// TIA Portal V17 export
// export: Created 2025-06-25T13:13:25.7107653Z, ExportSetting WithDefaults, DisplayName Totally Integrated Automation Portal, DisplayVersion V17 Update 8, DisplayName TIA Portal Openness, DisplayVersion V17 Update 8, DisplayName TIA Portal Version Control Interface, DisplayVersion V17, DisplayName STEP 7 Professional, DisplayVersion V17 Update 8, DisplayName STEP 7 Safety, DisplayVersion V17 Update 6, DisplayName WinCC Advanced, DisplayVersion V17 Update 8
DATA_BLOCK "DB_Application"   // DB9
{ S7_Optimized_Access := 'FALSE' }
VERSION : 0.1
// stored: AutoNumber true, DBAccessibleFromOPCUA true, DBAccessibleFromWebserver true, IsOnlyStoredInLoadMemory false, IsWriteProtectedInAS false
   VAR
      ToHB : Struct
         StartRequest : Bool;
         StopRequest : Bool;
         AlarmAcknowledge : Bool;
         EmergencyStopResetRequest : Bool;
         FastStopRequest : Bool;
         HydrolockProtection : Bool;
         SpareCommand6 : Bool;
         SpareCommand7 : Bool;
         SuperheatManualMode : Bool;
         HeatSinkOutManualMode : Bool;
         PerformanceControlManualMode : Bool;
         OilHeatingRegulatorManualMode : Bool;
         ExpansionValveRegulatorManualMode : Bool;
         PinchRegulatorManualMode : Bool;
         SpareManualMode6 : Bool;
         SpareManualMode7 : Bool;
         PumaCommOk : Bool;   // 1 = communication OK, 0 = communication dead
         HeatSourceOk : Bool;   // 1 = Source ready, 0 = source not ready
         HeatSinkOk : Bool;   // 1 = Sink ready, 0 = sink not ready
         SpareGroup2Command3 : Bool;
         SpareGroup2Command4 : Bool;
         SpareGroup2Command5 : Bool;
         SpareGroup2Command6 : Bool;
         SpareGroup2Command7 : Bool;
         SpareGroup3Command0 : Bool;
         SpareGroup3Command1 : Bool;
         SpareGroup3Command2 : Bool;
         SpareGroup3Command3 : Bool;
         SpareGroup3Command4 : Bool;
         SpareGroup3Command5 : Bool;
         SpareGroup3Command6 : Bool;
         SpareGroup3Command7 : Bool;
         SuperheatManualValue : Real;
         HeatSinkOutManualValue : Real;
         PerformanceControlManualValue : Real;
         OilHeatingManualValue : Real;
         ExpansionValveManualValue : Real;
         PinchManualValue : Real;
         HeatboosterSetpoint : Real;
         RegulationTarget : Int;
         LivenessCounter : UInt;
         HBL_HCV_514_A1 : Real;   // If externally controlled
         HBL_HCV_548_A1 : Real;   // If externally controlled
         HBL_TT_546 : Real;   // If externally controlled
         HBL_PT_547 : Real;   // If externally controlled
         HBL_HCV_515_A1 : Real;   // If externally controlled
         HBL_TT_901 : Real;   // If externally controlled
         HBL_PT_902 : Real;   // If externally controlled
         HBL_TT_512 : Real;   // If externally controlled
         HBL_PT_511 : Real;   // If externally controlled
         HBL_PT_519 : Real;   // If externally controlled
         HBL_TT_518 : Real;   // If externally controlled
      END_STRUCT;
      FromHB : Struct
         EmergencyStop : Bool;
         OilHeatersGroup1 : Bool;
         OilHeatersGroup2 : Bool;
         HBL_SC_01_Ready : Bool;
         HBL_SC_01_Run : Bool;
         HBL_SC_01_Tripped : Bool;
         HBL_SC_02_Ready : Bool;
         HBL_SC_02_Run : Bool;
         HBL_SC_02_Tripped : Bool;
         HBL_SC_10_Ready : Bool;
         HBL_SC_10_Run : Bool;
         HBL_SC_10_Tripped : Bool;
         HBL_HV_630 : Bool;
         HBL_HV_631 : Bool;
         HBL_HV_860 : Bool;
         HBL_HV_861 : Bool;
         HBL_HV_114 : Bool;
         HBL_HV_115 : Bool;
         CPC_P_01 : Bool;
         SSC_P_01 : Bool;
         SSC_F_01 : Bool;
         SSC_P_02 : Bool;
         HBL_LS_01 : Bool;
         HBL_LS_02 : Bool;
         HBL_HV_112 : Bool;
         HBL_HV_113 : Bool;
         HBL_LSH_62 : Bool;
         HBL_LSL_63 : Bool;
         HBL_LSH_64 : Bool;
         HBL_LSL_864 : Bool;
         HBL_LS_632 : Bool;
         HBL_LS_633 : Bool;
         HBL_SC_03_Ready : Bool;
         HBL_SC_03_Run : Bool;
         HBL_SC_03_Tripped : Bool;
         HBL_HCV_514_Force : Bool;
         HBL_HCV_548_Force : Bool;
         Spare05 : Bool;
         Spare06 : Bool;
         Spare07 : Bool;
         MachineState : Int;
         CompressorType : Int;
         SystemType : Int;
         RefrigerantType : Int;
         UptimeHours : Int;
         UptimeMinutes : Int;
         UptimeSeconds : Int;
         ActiveTimeHours : Int;
         ActiveTimeMinutes : Int;
         ActiveTimeSeconds : Int;
         RunningTimeHours : Int;
         RunningTimeMinutes : Int;
         RunningTimeSeconds : Int;
         Alarms : Array[0..159] of Bool;   // Compressed alarm bits
         HeatboosterSetpoint : Real;
         RegulationTarget : Int;
         HBL_HCV_514 : Real;   // Force setpoint
         HBL_HCV_548 : Real;   // Force setpoint
         DB_AI : Struct
            HBL_TT_502 : Real;
            HBL_PT_503 : Real;
            HBL_TT_504 : Real;
            HBL_LT_510 : Real;
            HBL_PT_511 : Real;
            HBL_TT_512 : Real;
            HBL_TT_516 : Real;
            HBL_PT_517 : Real;
            HBL_TT_518 : Real;
            HBL_PT_519 : Real;
            HBL_FT_520 : Real;
            HBL_TT_530 : Real;
            HBL_PT_531 : Real;
            HBL_TT_532 : Real;
            HBL_TT_533 : Real;
            HBL_PT_534 : Real;
            HBL_AT_535 : Real;
            HBL_TT_540 : Real;
            HBL_PT_541 : Real;
            HBL_TT_542 : Real;
            HBL_TT_543 : Real;
            HBL_PT_544 : Real;
            HBL_AT_545 : Real;
            HBL_TT_546 : Real;
            HBL_PT_547 : Real;
            HBL_TT_571 : Real;
            HBL_PT_572 : Real;
            HBL_TT_573 : Real;
            HBL_LT_610 : Real;
            HBL_TT_611 : Real;
            HBL_PT_612 : Real;
            HBL_CT_615 : Real;
            HBL_PT_618 : Real;
            HBL_PT_635 : Real;
            HBL_PT_636 : Real;
            HBL_LT_650 : Real;
            HBL_PT_651 : Real;
            HBL_PT_701 : Real;
            HBL_PT_702 : Real;
            HBL_PT_703 : Real;
            CPC_LT_870 : Real;
            CPC_TT_871 : Real;
            CPC_PT_872 : Real;
            CPC_PT_862 : Real;
            HBL_TT_901 : Real;
            HBL_PT_902 : Real;
            HBL_TT_03 : Real;
            HBL_TT_16 : Real;
            HBL_TT_17 : Real;
            HBL_TT_18 : Real;
            HBL_TT_20 : Real;
            HBL_TT_21 : Real;
            HBL_TT_22 : Real;
            HBL_TT_23 : Real;
            HBL_TT_24 : Real;
            HBL_TT_25 : Real;
            HBL_TT_26 : Real;
            HBL_TT_27 : Real;
            HBL_PT_05 : Real;
            HBL_PT_06 : Real;
            HBL_PT_17 : Real;
            HBL_CT_01 : Real;
            HBL_CT_03 : Real;
            SSC_TT_01 : Real;
            SSC_TT_02 : Real;
            SSC_TT_03 : Real;
            SSC_TT_04 : Real;
            SSC_PIT_01 : Real;
            SSC_PDT_01 : Real;
            SSC_LT_01 : Real;
         END_STRUCT;
         DB_Calc : Struct
            Compressor_CrankcaseSaturationTemperature : Real;
            Compressor_CrankcaseSuperheat : Real;
            Compressor_VolumetricEfficiency : Real;
            Compressor_IsentropicEfficiency : Real;
            Compressor_Massflow : Real;
            Heatsink_DeltaT : Real;
            Heatsink_Pinch : Real;
            Heatsink_Heatrate : Real;
            Heatsink_DeltaP : Real;
            Heatsink_Massflow : Real;
            Heatsource_DeltaT : Real;
            Heatsource_Pinch : Real;
            Heatsource_Heatrate : Real;
            Heatsource_DeltaP : Real;
            Heatsource_TemperatureRateOfChange : Real;
            Heatsource_Massflow : Real;
            HighPressPart_CompressorSaturationTemperature : Real;
            HighPressPart_CompressorSuperheat : Real;
            HighPressPart_CondenserSaturationTemperature : Real;
            HighPressPart_CondenserSubcooling : Real;
            HighPressPart_ExpansionValveSubcooling : Real;
            HighPressPart_CondenserDeltaP : Real;
            LowPressPart_EvaporatorSuperheat : Real;
            LowPressPart_CompressorSuperheat : Real;
            LowPressPart_EvaporatorSaturationTemperature : Real;
            LowPressPart_CompressorSaturationTemperature : Real;
            System_Quality : Real;
            System_COP : Real;
            System_ElectricalPower : Real;
            System_TemperatureLift : Real;
            System_MotorEfficiency : Real;
            System_FMEP : Real;
            Aux_ShaftSealDeltaT : Real;
            Aux_CPCPumpDeltaP : Real;
            Misc_EvaporatorDischargePressureMean : Real;
            Misc_EvaporatorDischargeTemperatureMin : Real;
            Misc_EvaporatorDischargeTemperatureMean : Real;
            Misc_OilFilterDeltaP : Real;
         END_STRUCT;
         DB_InverterDrives : Struct
            HBL_SC_01_A1 : Real;
            HBL_SC_01_A2 : Real;
            HBL_SC_01_A3 : Real;
            HBL_SC_02_A1 : Real;
            HBL_SC_02_A2 : Real;
            HBL_SC_02_A3 : Real;
            HBL_SC_10_A1 : Real;
            HBL_SC_10_A2 : Real;
            HBL_SC_10_A3 : Real;
            HBL_SC_03_A1 : Real;
            HBL_SC_03_A2 : Real;
            HBL_SC_03_A3 : Real;
         END_STRUCT;
         DB_Valves : Struct
            HBL_HCV_576_A1 : Real;
            HBL_HCV_578_A1 : Real;
            HBL_HCV_577_A1 : Real;
            HBL_HCV_579_A1 : Real;
            HBL_HCV_515_A1 : Real;
            HBL_HCV_575_A1 : Real;
            HBL_HCV_616_A1 : Real;
            HBL_HCV_700_A1 : Real;
            HBL_HCV_514_A1 : Real;
            HBL_HCV_548_A1 : Real;
         END_STRUCT;
      END_STRUCT;
   END_VAR
BEGIN
END_DATA_BLOCK
